FUNCTION EtapeEnCours : STRING(50)
VAR_INPUT
END_VAR
VAR
	icounter:INT;
END_VAR

FOR icounter := G_Match.iLigne TO 1 BY -1 DO
	IF G_Match.Tableau[G_Match.iCounter].NomEtape <> '' THEN
		EtapeEnCours := G_Match.Tableau[G_Match.iCounter].NomEtape;
		EXIT;
	END_IF
END_FOR

END_FUNCTION

(* stored: Version 1.1.0.1, ProductVersion 3.1.4024.12
   POU EtapeEnCours: Id {72cf8a31-bffd-4f0c-9dc6-ce14aa078678}, SpecialFunc None *)
